ABB RobotStudio station: Project3.rsstnx

Station Project3 (saved by RobotStudio 22.3.10141.1)
Controller Controlador1, task T_ROB1: task frame (RAPID world) sits at (824.5, 292, 460) mm in the station
Controller Controlador1
  mechanical unit ROB_1: IRB4600_20_250_C_01, 6 joints, base frame (0, 0, 0) mm
  mechanical unit TRACK_1: IRBT2005_IRB_STD_INT_0_0_2__01, 1 joints, base frame (0, 0, 0) mm
Layout (positions relative to the parent item):
  - IRB4600_20_250_C_01 [mechanism, from Robots\IRB4600_20_250_C_G_01.rslib] at (324.5, 292, 460) mm; joint values [0.7952, 0, 0, 0, 0.5236, 0] (rad or m)
  - IRBT2005_IRB_STD_INT_0_0_2__01 [mechanism] at (0, 0, 0) mm; joint values [-0.5] (rad or m)
      links: Base, Link1
Attachment: IRB4600_20_250_C_01 is attached to IRBT2005_IRB_STD_INT_0_0_2__01 / Link1
